// Mitsubishi GX Works2 project: first_study   PLC: FX3U/FX3UC

PROGRAM MAIN
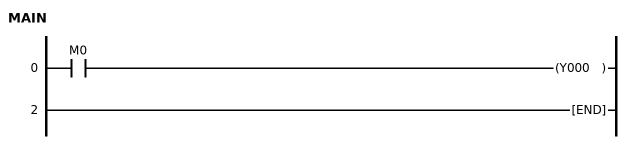
0     LD      M0
      OUT     Y000
2     END
END_PROGRAM
